(* IEC 61131-3 sources: AXOpen/src/components.siemens.identification/app/SystemConstants, 2 files *)

(* ---- plc_line_HwIdentifiers.st ---- *)
CONFIGURATION HardwareIDs
    VAR_GLOBAL CONSTANT
        et200sp_CM_4xIO_Link_RF200_HwID : UINT := UINT#260;
        et200sp_CM_4xIO_Link_RF200_CM_4xIO_Link_V2_2_144I_128O_1_CM_4xIO_Link_V2_2_144I_128O_HwID : UINT := UINT#264;
        et200sp_CM_4xIO_Link_RF200_Rack_HwID : UINT := UINT#261;
        et200sp_CM_4xIO_Link_RF200_Server_module_V1_1_Server_module_V1_1_0_bytes_HwID : UINT := UINT#263;
        et200sp_CM_4xIO_Link_RF200_et200sp_CM_4xIO_Link_RF200_HwID : UINT := UINT#262;
        et200sp_CM_4xIO_Link_RF200_et200sp_CM_4xIO_Link_RF200_IM_155_6_PN_ST_V4_2_HwID : UINT := UINT#265;
        et200sp_CM_4xIO_Link_RF200_et200sp_CM_4xIO_Link_RF200_Port_1_HwID : UINT := UINT#258;
        et200sp_CM_4xIO_Link_RF200_et200sp_CM_4xIO_Link_RF200_Port_2_HwID : UINT := UINT#259;
        et200sp_CM_4xIO_Link_RF200_et200sp_CM_4xIO_Link_RF200_profinet_HwID : UINT := UINT#257;
        plc_line_HwID : UINT := UINT#32;
        plc_line_Rail_0_HwID : UINT := UINT#275;
        plc_line_plc_line_HwID : UINT := UINT#48;
        plc_line_plc_line_CPU_display_1_HwID : UINT := UINT#54;
        plc_line_plc_line_Card_reader_writer_1_HwID : UINT := UINT#51;
        plc_line_plc_line_DP_interface_1_HwID : UINT := UINT#60;
        plc_line_plc_line_OPC_UA_1_HwID : UINT := UINT#117;
        plc_line_plc_line_profinet_x1_HwID : UINT := UINT#64;
        plc_line_plc_line_profinet_x1_Port_1_HwID : UINT := UINT#65;
        plc_line_plc_line_profinet_x1_Port_2_HwID : UINT := UINT#66;
        plc_line_plc_line_profinet_x2_HwID : UINT := UINT#72;
        plc_line_plc_line_profinet_x2_Port_3_HwID : UINT := UINT#73;
        plc_line_plc_line_virtual_communication_interface_HwID : UINT := UINT#135;
        profinet_plc_line_HwID : UINT := UINT#256;
        rf186c_HwID : UINT := UINT#269;
        rf186c_Rack_HwID : UINT := UINT#270;
        rf186c_Reader_1__Reader__HwID : UINT := UINT#272;
        rf186c_rf186c_HwID : UINT := UINT#271;
        rf186c_rf186c_CM_1__Communication__HwID : UINT := UINT#273;
        rf186c_rf186c_RF186C___V2_x_HwID : UINT := UINT#274;
        rf186c_rf186c_profinet_HwID : UINT := UINT#266;
        rf186c_rf186c_profinet_Port_1_HwID : UINT := UINT#267;
        rf186c_rf186c_profinet_Port_2_HwID : UINT := UINT#268;

    END_VAR
END_CONFIGURATION

(* ---- plc_line_IoAddresses.st ---- *)
CONFIGURATION IoAddresses
    VAR_GLOBAL
        et200sp_CM_4xIO_Link_V2_2_144I_128O_1_InputAddress_0 AT %IL0: LWORD;
        et200sp_CM_4xIO_Link_V2_2_144I_128O_1_InputAddress_1 AT %IL8: LWORD;
        et200sp_CM_4xIO_Link_V2_2_144I_128O_1_InputAddress_2 AT %IL16: LWORD;
        et200sp_CM_4xIO_Link_V2_2_144I_128O_1_InputAddress_3 AT %IL24: LWORD;
        et200sp_CM_4xIO_Link_V2_2_144I_128O_1_InputAddress_4 AT %IL32: LWORD;
        et200sp_CM_4xIO_Link_V2_2_144I_128O_1_InputAddress_5 AT %IL40: LWORD;
        et200sp_CM_4xIO_Link_V2_2_144I_128O_1_InputAddress_6 AT %IL48: LWORD;
        et200sp_CM_4xIO_Link_V2_2_144I_128O_1_InputAddress_7 AT %IL56: LWORD;
        et200sp_CM_4xIO_Link_V2_2_144I_128O_1_InputAddress_8 AT %IL64: LWORD;
        et200sp_CM_4xIO_Link_V2_2_144I_128O_1_InputAddress_9 AT %IL72: LWORD;
        et200sp_CM_4xIO_Link_V2_2_144I_128O_1_InputAddress_10 AT %IL80: LWORD;
        et200sp_CM_4xIO_Link_V2_2_144I_128O_1_InputAddress_11 AT %IL88: LWORD;
        et200sp_CM_4xIO_Link_V2_2_144I_128O_1_InputAddress_12 AT %IL96: LWORD;
        et200sp_CM_4xIO_Link_V2_2_144I_128O_1_InputAddress_13 AT %IL104: LWORD;
        et200sp_CM_4xIO_Link_V2_2_144I_128O_1_InputAddress_14 AT %IL112: LWORD;
        et200sp_CM_4xIO_Link_V2_2_144I_128O_1_InputAddress_15 AT %IL120: LWORD;
        et200sp_CM_4xIO_Link_V2_2_144I_128O_1_InputAddress_16 AT %IL128: LWORD;
        et200sp_CM_4xIO_Link_V2_2_144I_128O_1_InputAddress_17 AT %IL136: LWORD;
        et200sp_CM_4xIO_Link_V2_2_144I_128O_1_OutputAddress_0 AT %QL0: LWORD;
        et200sp_CM_4xIO_Link_V2_2_144I_128O_1_OutputAddress_1 AT %QL8: LWORD;
        et200sp_CM_4xIO_Link_V2_2_144I_128O_1_OutputAddress_2 AT %QL16: LWORD;
        et200sp_CM_4xIO_Link_V2_2_144I_128O_1_OutputAddress_3 AT %QL24: LWORD;
        et200sp_CM_4xIO_Link_V2_2_144I_128O_1_OutputAddress_4 AT %QL32: LWORD;
        et200sp_CM_4xIO_Link_V2_2_144I_128O_1_OutputAddress_5 AT %QL40: LWORD;
        et200sp_CM_4xIO_Link_V2_2_144I_128O_1_OutputAddress_6 AT %QL48: LWORD;
        et200sp_CM_4xIO_Link_V2_2_144I_128O_1_OutputAddress_7 AT %QL56: LWORD;
        et200sp_CM_4xIO_Link_V2_2_144I_128O_1_OutputAddress_8 AT %QL64: LWORD;
        et200sp_CM_4xIO_Link_V2_2_144I_128O_1_OutputAddress_9 AT %QL72: LWORD;
        et200sp_CM_4xIO_Link_V2_2_144I_128O_1_OutputAddress_10 AT %QL80: LWORD;
        et200sp_CM_4xIO_Link_V2_2_144I_128O_1_OutputAddress_11 AT %QL88: LWORD;
        et200sp_CM_4xIO_Link_V2_2_144I_128O_1_OutputAddress_12 AT %QL96: LWORD;
        et200sp_CM_4xIO_Link_V2_2_144I_128O_1_OutputAddress_13 AT %QL104: LWORD;
        et200sp_CM_4xIO_Link_V2_2_144I_128O_1_OutputAddress_14 AT %QL112: LWORD;
        et200sp_CM_4xIO_Link_V2_2_144I_128O_1_OutputAddress_15 AT %QL120: LWORD;
        rf186c_CM_1_InputAddress AT %IW146: WORD;
        rf186c_CM_1_OutputAddress AT %QW130: WORD;
        rf186c_Reader_1_InputAddress AT %IW144: WORD;
        rf186c_Reader_1_OutputAddress AT %QW128: WORD;

    END_VAR
END_CONFIGURATION
